Universal Robots PolyScope program: mecspe_refactor2.urp

Program mecspe_refactor2 (installation=mecspe_install directory=/home/ur/ursim-current/programs/mecspe2 createdIn=3.15.4.106291 lastSavedIn=3.15.4.106291 robotSerialNumber=2018359999)
Calibrated DH parameters: a=[0.000104, -0.381245, -0.385946, 0.00002, 0.000083, 0]; d=[0.089177, 59.99214, -36.297918, -23.584132, 0.094784, 0.082552]; alpha=[1.570197, -0.003145, 0.002952, 1.570494, -1.570091, 0]; deltaTheta=[-0.00001, -0.459739, 0.638868, -0.17972, -0.000006, -0.000462]
InitVariablesNode variables(variable(name=nCycle, expression=0), variable(name=stock, expression=[16,16,16,40,16,16,16,40,16,16,16,40,16,40,0,0,0,0,0,0,0,0,0,0]))
BeforeStart
  Script file /home/ur/ursim-current/programs/mecspe2/calc_pose_to_position.script
    | def calc_pose_to_position(pose, feature, position):
    | 
    |    PoseRelativeToFeature = pose_trans(pose_inv(feature), pose)
    | 
    |    diff = pose_sub(position, PoseRelativeToFeature)
    |    vect = p[diff[0], diff[1], diff[2], 0, 0, 0]
    | 
    |    MoveTCPRelativeToFeature = pose_add(PoseRelativeToFeature, vect)
    |    return pose_trans(feature, MoveTCPRelativeToFeature)
    | 
    | end
  Script file /home/ur/ursim-current/programs/mecspe2/calc_item_position.script
    | def calc_item_position(item, prop, grid, module, seat, compens):
    | 
    |     # calcola la posizione assoluta del pezzo scelto da pickPalletItem
    | 
    |     # nPosX è il numero di colonne
    |     # nPosY è il numero di righe
    |     # distX è la distanza tra colonne
    |     # distY è la distanza tra righe
    |     # [posX1, posY1] è la posizione del primo pezzo rispetto all'origine del pallet
    | 
    |     nPallet = module # module e seat partono da 1
    |     nItem = seat
    | 
    |     nPosXgrid = grid[0] # numero di posizioni della giglia in X
    |     distXgrid = grid[2] # distanza tra gli slot della griglia in X
    |     distYgrid = grid[3] # distanza tra gli slot della griglia in Y
    | 
    |     pallPosX = nPallet%nPosXgrid
    |     if(pallPosX==0): pallPosX = nPosXgrid end
    |     pallPosY = ceil(nPallet/nPosXgrid)
    | 
    |     pallPosX1 = grid[4]
    |     pallPosY1 = grid[5]
    | 
    | 
    |     nPosX = prop[item,0]
    |     nPosY = prop[item,1]
    |     distX = prop[item,2]
    |     distY = prop[item,3]
    |     posX1 = prop[item,4]
    |     posY1 = prop[item,5]
    | 
    |     posX = nItem%nPosX
    |     if(posX==0): posX = nPosX end
    |     posY = ceil(nItem/nPosX)
    | 
    |     position = p[0,0,0,0,0,0]
    | 
    |     X=distX*(posX - 1) + posX1 + distXgrid*(pallPosX - 1) + pallPosX1 + compens[0]*1000
    |     Y=distY*(posY - 1) + posY1 + distYgrid*(pallPosY - 1) + pallPosY1 + compens[1]*1000
    | 
    |     position[0] = X/1000
    |     position[1] = Y/1000
    | 
    |     return position
    | 
    |  end
  Script file /home/ur/ursim-current/programs/mecspe2/calc_compens_pos.script
    | def calc_compens_pos(item, prop, grid, module, feature, posAppr):
    | 
    | 	compens = p[0,0,0,0,0,0]
    | 	posPred = calc_item_position(item, prop, grid, module, 1, compens)
    | 
    | 	posApprFeat = pose_trans(pose_inv(feature), posAppr)
    | 	diff = pose_sub(posApprFeat,posPred)
    | 
    | 	compens[0] = diff[0]
    | 	compens[1] = diff[1]
    | 
    | 	return compens
    | 
    | end
  Script file /home/ur/ursim-current/programs/mecspe2/tcpMov.script
    | def tcpMov(vect):
    | 
    |     # FeaturePose is the pose for the feature
    |     # vect = p[0.1, 0, 0, 0, 0, 0] makes us move 10cm in the X direction of the feature
    |     # credits: https://forum.universal-robots.com/t/move-tcp-relative-to-feature/15492
    | 
    |    tcp_pose = get_actual_tcp_pose()
    |    return pose_add(tcp_pose, vect)
    | 
    | 
    | end
  Script file /home/ur/ursim-current/programs/mecspe2/gen_tcp_grid.script
    | def next_tcp_grid_pos(cur_pos,size,dist):
    | 
    | # size e' la dimensione della griglia da generare,
    | # 2 significa 2x2, 3 significa 3x3 etc
    | 
    | rel_p = [0,0]
    | tcpp = get_actual_tcp_pose()
    | 
    | posX = cur_pos%size
    | if(posX==0): posX = size end
    | posY = ceil(cur_pos/size)
    | 
    | actual_dx = -dist*(size-1)/2 + (posX-1)*dist
    | actual_dy= -dist*(size-1)/2 + (posY-1)*dist
    | 
    | posX = (cur_pos+1)%size
    | if(posX==0): posX = size end
    | posY = ceil((cur_pos+1)/size)
    | 
    | next_dx = -dist*(size-1)/2 + (posX-1)*dist
    | next_dy= -dist*(size-1)/2 + (posY-1)*dist
    | 
    | rel_p = [next_dx - actual_dx, next_dy - actual_dy]
    | 
    | return rel_p
    | 
    | end
  Script file /home/ur/ursim-current/programs/andrea11/stock_update.script
    | def stock_update(modulo_posto,stock):
    | 
    |     i = modulo_posto[0]
    |     stock[i] = stock[i] - 1
    |     return stock
    | 
    | 
    | end
  Script file /home/ur/ursim-current/programs/mecspe2/select_module_seat.script
    | def select_module_seat(type, properties, layout, stocks):
    | 
    |   if type < 0:
    |       request_integer_from_primary_client("Tipo di oggetto selezionato non specificato. specificare oggetto")
    |   end
    | 
    | 
    |   # seleziona un pezzo sulla griglia, noti il tipo di pezzo e lo stato della griglia
    | 
    |   # lo script funziona finché le variabili del robot non vengono resettate. Tuttavia, anche
    |   # in caso di riavvio, è possibile scrivere manualmente le info sulla griglia e lo stock
    |   # all'inizio del programma, così da 'insegnare' al robot dove farlo
    |   # riprendere
    | 
    |   iPallet = 0 # inizializzo l'id del pallet
    | 
    |   while iPallet < length(layout):
    | 
    |     if layout[iPallet] == type and stocks[iPallet] > 0 :
    | 
    |       nItems = stocks[iPallet] # numero di pezzi nello stock del pallet iesimo
    | 
    |       nPosX = properties[type,0] # numero di posizioni lungo x, come definito per il pallet di tipo "type"
    |       nPosY = properties[type,1] # numero di posizioni lungo y, come definito per il pallet di tipo "type"
    | 
    |       stockMax = nPosX*nPosY
    |       iItem = stockMax - nItems # id del pezzo
    | 
    |       nPallet = iPallet + 1
    |       nItem = iItem + 1
    | 
    |       nModuloPosto = [nPallet,nItem]
    | 
    |       # nModuloPosto = [numero del pallet, numero del posto sul pallet]
    | 
    |       return nModuloPosto
    |  end
    | iPallet = iPallet + 1
    | end
    | end
  Script file /home/ur/ursim-current/programs/mecspe2/ini_grid.script
    | def ini_grid():
    | 
    |     # grid = [nPallPosX, nPallPosY, distPallX, distPallY, pallPosX1, pallPosY1, pallPosZ1]
    |     # la struttura e' del tutto analoga in logica con quella espressa in defs
    |     grid = [4, 6, 90, 90, 10, 20, 6]
    |     return grid
    | end
  Script file /home/ur/ursim-current/programs/mecspe2/ini_properties.script
    | chp = 1
    | ghr = 2
    | 
    | def ini_properties():
    | 
    |     # definition = [nPosX,nPosY,distX,distY,posX1,posY1,posZ1]
    | 
    |     # nPosX è il numero di colonne
    |     # nPosY è il numero di righe
    |     # distX è la distanza tra colonne
    |     # distY è la distanza tra righe
    |     # [posX1, posY1] è la posizione del primo pezzo rispetto all'origine del pallet
    |     # posZ1 e' la posizione che deve raggiungere il TCP lungo asse Z, che sarebbe asse verticale
    | 
    |     prop = [
    |         [0, 0, 0, 0, 0, 0, 0], # slot vuoto
    |         [4, 10, 18, 8, 17, 10.3, 10], # pallet chip
    |         [4, 4, 21, 21, 12.5, 12.5, 50], # pallet ghiere
    |         [1, 1, 0, 0, 132.06, 44, 16.05], # stazione antenna
    |         [1, 2, 0, 40, 20.256, 24, 27.85], # stazione incollaggio
    |         [1, 1, 0, 0, 40, 40, 50] # cestino
    |     ]
    |     return prop
    | end
  Script file /home/ur/ursim-current/programs/mecspe2/ini_layout.script
    | def ini_layout():
    | 
    |     visualLayout = [
    | 
    |         [0, 0, 0, 0],
    |         [0, 0, 0, 0],
    |         [0,0,0,0],
    |         [0,0,0,0],
    |         [0,ghr,0,chp],
    |         [0,0,0,0]
    | 
    |     ]
    | 
    | # purtroppo fare questa array vuota di dimensione (righe)x(colonne) per aggirare le limitazioni di UR
    | # bisogna ricordarsi di cambiare questa dichiarazione di types se si cambia dimensione griglia
    | 
    |      layout = [0,0,0,0,0,0,0,0,0,0,0,0,0,0,0,0,0,0,0,0,0,0,0,0]
    | 
    |     iii = 0
    |     s = size(visualLayout)
    |     i = 0
    |     while i < s[0]:
    | 
    |         ii=0
    |         while ii < s[1]:
    | 
    |             layout[iii] = visualLayout[s[0]-1-i,ii]
    |             ii = ii + 1
    |             iii = iii + 1
    |         end
    |     i = i + 1
    |     end
    |     return layout
    | end
  Script file /home/ur/ursim-current/programs/mecspe2/ini_stocks.script
    | def ini_stocks(defs, types):
    | 
    |     global f = -1 # usa questo carattere per inizializzare automaticamente pallet pieni
    | 
    |     visualStocks = [
    | 
    |         [f, f, f, f],
    |         [f, f, f, f],
    |         [f, f, f, f],
    |         [f, f, f, f],
    |         [f, f, f, f],
    |         [f ,f, f, f]
    | 
    |     ]
    | 
    | # purtroppo occorre fare questa array vuota di dimensione (righe)x(colonne) per aggirare le limitazioni di UR
    | # bisogna ricordarsi di cambiare questa dichiarazione di types se si cambia dimensione griglia
    | 
    |      stocks = [0,0,0,0,0,0,0,0,0,0,0,0,0,0,0,0,0,0,0,0,0,0,0,0]
    | 
    |     iii = 0
    |     s = size(visualStocks)
    |     i = 0
    |     while i < s[0]:
    | 
    |         ii=0
    |         while ii < s[1]:
    |             if visualStocks[s[0]-1-i,ii] == f:
    |                 nPosX = defs[types[iii], 0]
    |                 nPosY = defs[types[iii], 1]
    |                 stocks[iii] = nPosX*nPosY
    |             else:
    | 
    |                 stocks[iii] = visualStocks[s[0]-1-i,ii]
    |             end
    |             ii = ii + 1
    |             iii = iii + 1
    |         end
    |     i = i + 1
    |     end
    |     return stocks
    | end
  Script file /home/ur/ursim-current/programs/mecspe2/fun_tens_utensile.script
    | def fun_tens_utensile():
    | 
    | 	i = 0
    | 	# invia 3 "impulsi" alla macchina per assicurarsi che il tool abbia tensione
    | 	while i < 3:
    | 		set_tool_voltage(24)
    | 		sleep(0.24)
    | 		i = i + 1
    | 	end
    | 
    | end
  Script file /home/ur/ursim-current/programs/mecspe2/ini_var.script
    | nModPosAttual = [
    | 
    | 	[0,0],
    | 	[0,0],
    | 	[0,0],
    | 	[0,0]
    | 
    | ]
    | 
    | nModPosPrec = [
    | 
    | 	[0,0],
    | 	[0,0],
    | 	[0,0],
    | 	[0,0]
    | 
    | ]
    | 
    | modulo_posto = [0,0]
  pose_apprend := get_actual_tcp_pose()
  statoPinza := 0
  statoGhiera := 0
  statoChip := 0
  compens := p[0,0,0,0,0,0]
  Set DigitalOutput pin=DO_ventosaOff; digitalValue=1
  Set DigitalOutput pin=DO_ventosaOn; digitalValue=0
  Set DigitalOutput pin=digital_out[2]; digitalValue=0
  layout := ini_layout()
  bypassVerifChp := False
  grid := ini_grid()
  properties := ini_properties()
  stock := ini_stocks(properties,layout)
  nCycle := 1
  chp_check := False
  Script: fun_tens_utensile()
  Wait Sleep waitTime=1
  testing := True
  Timer (action=Start) variable(name=timer_1)
  apprendimento := False
Robot Program (runOnlyOnce=false)
  If testing≟ True
    Call prel_ghr_pall
  SuppressedNode
    Else 
      MoveJ speed 60 deg/s, acceleration 80 deg/s^2 (useActiveTCP=true)
        Waypoint Waypoint_7: TCP in base x=321.623 y=412.075 z=-71.725 mm, rx=1.5831 ry=-2.4822 rz=0.1268 rad; joints [-138.339, -65.21, 105.073, -118.045, -93.062, 36.92] deg; flange x=345.08 y=447.244 z=123.756 mm, rx=2.1618 ry=-1.9789 rz=0.0478 rad
      selezione := ghr
      Call prel_ghr_pall
      statoGhiera := 1
      stock := stock_update(modulo_posto,stock)
      Call depo_ghr_col
      statoGhiera := 2
      chp_check := False
      Loop While (checkContinuously=false) expression=chp_check≟ False
        selezione := chp
        Call prel_chp_pall
        statoChip := 1
        MoveJ speed 60 deg/s, acceleration 80 deg/s^2 (useActiveTCP=false) tcp=Ventosa
          Waypoint Punto_percors_1: TCP in base x=331.541 y=425.449 z=-23.301 mm, rx=1.7621 ry=-0.7398 rz=-1.7726 rad; joints [-145.076, -38.163, 77.174, -38.938, -53.96, -45.259] deg; flange x=377.019 y=458.221 z=10.448 mm, rx=1.7621 ry=-0.7398 rz=-1.7726 rad
        Call seq_chp_ant
        If chp_check≟ True
          Call dosa_ades_col
          Call pressa_nfc_col
          Call prel_ghr_col
        Else 
          Call depo_chp_pal
Thread Thread_1 (runOnlyOnce=false)
  If timer_1>4
    Timer (action=Reset) variable=timer_1
    Script: fun_tens_utensile()
    Timer (action=Start) variable=timer_1
SubProgram -> prel_ghr_pall
SubProgram  [hidden by the author, left out]
SubProgram  [hidden by the author, left out]
SubProgram depo_ghr_pall [hidden by the author, left out]
SubProgram  [hidden by the author, left out]
SubProgram  [hidden by the author, left out]
SubProgram  [hidden by the author, left out]
SubProgram  [hidden by the author, left out]
SubProgram  [hidden by the author, left out]
SubProgram prel_ghr_pall (keepSynchronizedWithDisk=false)
  oggetto := ghr
  pose_apprend := pose_appPallGhr
  If apprendimento≟ True
    MoveJ speed 60 deg/s, acceleration 80 deg/s^2 (useActiveTCP=false) tcp=Pinza
      Waypoint pose_appPallGhr referenceName=pose_appPallGhr: TCP in base x=141.508 y=430.186 z=-147.75 mm, rx=0.607 ry=-1.4882 rz=-0.6293 rad; joints [-125.755, -39.244, 81.167, -41.963, -34.571, 44.831] deg; flange x=189.515 y=570.182 z=1.456 mm, rx=0.607 ry=-1.4882 rz=-0.6293 rad
      modulo :=  (valueSource=Operator message=Specificare il numero di modulo usato per l'apprendimento valueType=Integer)
      compens := calc_compens_pos(oggetto,properties,grid,modulo,piano_moduli,pose_apprend)
      Popup Message (haltProgram=false inputType=Variable) variable=compens
  Else 
    MoveJ speed 60 deg/s, acceleration 80 deg/s^2 (useActiveTCP=false) tcp=Pinza
      compens := p[0,0,0,0,0,0]
      nModuloPosto := select_module_seat(oggetto,properties,layout,stock)
      posizione := calc_item_position(oggetto,properties,grid,nModuloPosto[0],nModuloPosto[1],compens)
      pose_pallettiz := calc_pose_to_position(pose_apprend, piano_moduli, posizione)
      Waypoint Waypoint (Variable): variable=pose_pallettiz
  MoveL speed 250 mm/s, acceleration 1200 mm/s^2 (useActiveTCP=false) tcp=Pinza; feature=Base
    Waypoint Waypoint_1 (Relative): relativeFromPosition TCP in base x=143.961 y=537.139 z=34.835 mm, rx=0.607 ry=-1.4882 rz=-0.6293 rad; joints [-125.506, -39.287, 81.209, -42.035, -34.619, 44.824] deg; TCP in base x=143.457 y=501.955 z=-0.687 mm, rx=0.607 ry=-1.4882 rz=-0.6293 rad; joints [-127.449, -38.931, 87.822, -48.999, -36.562, 44.817] deg; flange x=189.012 y=534.998 z=-34.066 mm, rx=0.607 ry=-1.4882 rz=-0.6293 rad
  MoveL speed 50 mm/s, acceleration 100 mm/s^2 (useActiveTCP=false) tcp=Pinza; feature=Base
    Waypoint Waypoint_2 (Relative): relativeFromPosition TCP in base x=143.457 y=501.955 z=-0.687 mm, rx=0.607 ry=-1.4882 rz=-0.6293 rad; joints [-127.449, -38.931, 87.822, -48.999, -36.562, 44.817] deg; TCP in base x=143.286 y=489.992 z=-12.765 mm, rx=0.607 ry=-1.4882 rz=-0.6293 rad; joints [-128.156, -38.626, 89.864, -51.344, -37.269, 44.815] deg; flange x=188.841 y=523.035 z=-46.144 mm, rx=0.607 ry=-1.4882 rz=-0.6293 rad
    SuppressedNode
      Script: tool()
    Waypoint Waypoint_3 (Relative): relativeFromPosition TCP in base x=143.286 y=489.992 z=-12.765 mm, rx=0.607 ry=-1.4882 rz=-0.6293 rad; joints [-128.156, -38.626, 89.864, -51.344, -37.269, 44.815] deg; TCP in base x=143.457 y=501.955 z=-0.687 mm, rx=0.607 ry=-1.4882 rz=-0.6293 rad; joints [-127.449, -38.931, 87.822, -48.999, -36.562, 44.817] deg; flange x=189.012 y=534.998 z=-34.066 mm, rx=0.607 ry=-1.4882 rz=-0.6293 rad
  MoveL speed 250 mm/s, acceleration 1200 mm/s^2 (useActiveTCP=false) tcp=Pinza; feature=Base
    Waypoint Waypoint_4 (Relative): relativeFromPosition TCP in base x=143.457 y=501.955 z=-0.687 mm, rx=0.607 ry=-1.4882 rz=-0.6293 rad; joints [-127.449, -38.931, 87.822, -48.999, -36.562, 44.817] deg; TCP in base x=143.961 y=537.139 z=34.835 mm, rx=0.607 ry=-1.4882 rz=-0.6293 rad; joints [-125.506, -39.287, 81.209, -42.035, -34.619, 44.824] deg; flange x=189.515 y=570.182 z=1.456 mm, rx=0.607 ry=-1.4882 rz=-0.6293 rad
SubProgram depo_ghr_col [hidden by the author, left out]
SubProgram prel_chp_pall [hidden by the author, left out]
SubProgram seq_chp_ant [hidden by the author, left out]
SubProgram dosa_ades_col [hidden by the author, left out]
SubProgram pressa_nfc_col [hidden by the author, left out]
SubProgram prel_ghr_col [hidden by the author, left out]
SubProgram depo_chp_pal [hidden by the author, left out]
